(* IEC 61131-3 sources: volt/packages/volt-lsp-iec/test-corpus/bakon-nano/Device/Plc Logic/Application/POUs/HMI Functions, 3 files *)

(* ---- RecipeChoiceSelector.pou ---- *)
PROGRAM RecipeChoiceSelector
VAR
	nOldClmn1Choice : INT;
	nOldClmn2Choice : INT;
	bChoiceSetToZero : BOOL;
END_VAR

%LANGUAGE ST
/////////// First Column ////////////////////////////////////////////////////////////////////////////////
(*
Choices:
SlabRound = 1
SlabRound with fingers = 2
Tray = 3
*)

IF g_HMI_MachCommand.CMD.bNewRecipe AND NOT bChoiceSetToZero THEN
	g_sHMI_Recipe_Clmn1_Choice := 0;
	g_sHMI_Recipe_Clmn2_Choice := 0;
	g_sHMI_Recipe_Clmn2_Choice := 0;
	bChoiceSetToZero := TRUE;
END_IF
IF NOT(g_HMI_MachCommand.CMD.bNewRecipe) THEN
	bChoiceSetToZero := FALSE;
END_IF
g_sHMI_RcpClmns.clmn1.SlabRound := gProductOption.Prod_RoundQuatro
								OR gProductOption.Prod_SlabDiagonal
								OR gProductOption.Prod_SlabSquare
								OR gProductOption.Prod_SlabDouble
								OR gProductOption.Prod_SlabTriangle;

g_sHMI_RcpClmns.clmn1.SlabRoundFngrs := gProductOption.Prod_Round
									OR gProductOption.Prod_SlabSquareClamp;

g_sHMI_RcpClmns.clmn1.Tray := gProductOption.Prod_TraySquareDouble
								OR gProductOption.Prod_TraySquareLarge
								OR gProductOption.Prod_TraySquareSmall
								OR gProductOption.Prod_TraySquareTriple;

(*Reset choice for clmn 2 and 3 when 1 is changed *)
IF nOldClmn1Choice <> g_sHMI_Recipe_Clmn1_Choice THEN
	g_sHMI_Recipe_Clmn2_Choice := 0;
	g_sHMI_Recipe_Clmn3_Choice := 0;
	nOldClmn1Choice := g_sHMI_Recipe_Clmn1_Choice;
END_IF

//////////////////////////////////////////////////////////////////////////////////////////////////////////

/////////// Second Column ////////////////////////////////////////////////////////////////////////////////
(*
Choises:
Slab= 1
Slab with Fingers = 2
Round = 3
Round with fingers = 4
Tray Small = 5
Tray Large = 6
Tray double = 7
Tray Quadruple = 8
*)
g_sHMI_RcpClmns.clmn2.Slab := (gProductOption.Prod_SlabDiagonal
								OR gProductOption.Prod_SlabSquare
								OR gProductOption.Prod_SlabDouble
								OR gProductOption.Prod_SlabTriangle)
								AND (g_sHMI_Recipe_Clmn1_Choice = 1);

g_sHMI_RcpClmns.clmn2.SlabFingers := gProductOption.Prod_SlabSquareClamp AND (g_sHMI_Recipe_Clmn1_Choice = 2);

g_sHMI_RcpClmns.clmn2.Round := gProductOption.Prod_RoundQuatro AND (g_sHMI_Recipe_Clmn1_Choice = 1);

g_sHMI_RcpClmns.clmn2.RoundFingers := gProductOption.Prod_Round AND (g_sHMI_Recipe_Clmn1_Choice = 2 );

g_sHMI_RcpClmns.clmn2.TraySmall := gProductOption.Prod_TraySquareSmall AND (g_sHMI_Recipe_Clmn1_Choice = 3 );

g_sHMI_RcpClmns.clmn2.TrayLarge := gProductOption.Prod_TraySquareLarge AND (g_sHMI_Recipe_Clmn1_Choice = 3 );

g_sHMI_RcpClmns.clmn2.TrayQuadruple := gProductOption.Prod_TraySquareTriple AND (g_sHMI_Recipe_Clmn1_Choice = 3 );

g_sHMI_RcpClmns.clmn2.TrayDouble := gProductOption.Prod_TraySquareDouble AND (g_sHMI_Recipe_Clmn1_Choice = 3 );;

(*Reset choice for clmn 3 when 2 is changed *)
IF nOldClmn2Choice <> g_sHMI_Recipe_Clmn2_Choice THEN
	g_sHMI_Recipe_Clmn3_Choice := 0;
	nOldClmn2Choice := g_sHMI_Recipe_Clmn2_Choice;
END_IF
//////////////////////////////////////////////////////////////////////////////////////////////////////////

/////////// Third Column ////////////////////////////////////////////////////////////////////////////////
(*
Choices:
Square = 1
Round = 2
Diagonal = 3
*)
g_sHMI_RcpClmns.clmn3.Square := (gProductOption.Prod_SlabSquare
								OR gProductOption.Prod_TraySquareDouble
								OR gProductOption.Prod_TraySquareLarge
								OR gProductOption.Prod_TraySquareSmall
								OR gProductOption.Prod_TraySquareTriple
								OR gProductOption.Prod_SlabSquareClamp)
								AND (g_sHMI_Recipe_Clmn2_Choice <> 3)
								AND (g_sHMI_Recipe_Clmn2_Choice <> 4)
								AND (g_sHMI_Recipe_Clmn2_Choice <> 0);

g_sHMI_RcpClmns.clmn3.Triangle := (gProductOption.Prod_SlabSquare
								OR gProductOption.Prod_TraySquareLarge
								OR gProductOption.Prod_SlabSquareClamp)
								AND (g_sHMI_Recipe_Clmn2_Choice <> 2)
								AND (g_sHMI_Recipe_Clmn2_Choice <> 3)
								AND (g_sHMI_Recipe_Clmn2_Choice <> 4)
								AND (g_sHMI_Recipe_Clmn2_Choice <> 0);

g_sHMI_RcpClmns.clmn3.Diagonal := (gProductOption.Prod_SlabSquare
								OR gProductOption.Prod_SlabSquareClamp)
								AND (g_sHMI_Recipe_Clmn2_Choice <> 2)
								AND (g_sHMI_Recipe_Clmn2_Choice <> 3)
								AND (g_sHMI_Recipe_Clmn2_Choice <> 4)
								AND (g_sHMI_Recipe_Clmn2_Choice <> 0);

//////////////////////////////////////////////////////////////////////////////////////////////////////////

//////////select correct product in recipe////////////////////////////////////////////////////////////////
IF (g_sHMI_Recipe_Clmn1_Choice = 1) AND (g_sHMI_Recipe_Clmn2_Choice = 1) AND (g_sHMI_Recipe_Clmn3_Choice = 1) THEN
	g_HMI_RCP_Parameters_Visu.nProductType := Prod_Slab_Rectangle_1x1;
ELSIF (g_sHMI_Recipe_Clmn1_Choice = 1) AND (g_sHMI_Recipe_Clmn2_Choice = 1) AND (g_sHMI_Recipe_Clmn3_Choice = 2) THEN
	g_HMI_RCP_Parameters_Visu.nProductType := Prod_Slab_Triangle_1x1;
ELSIF (g_sHMI_Recipe_Clmn1_Choice = 1) AND (g_sHMI_Recipe_Clmn2_Choice = 1) AND (g_sHMI_Recipe_Clmn3_Choice = 3) THEN
	g_HMI_RCP_Parameters_Visu.nProductType := Prod_Slab_Diagonal_1x1;
ELSIF (g_sHMI_Recipe_Clmn1_Choice = 2) AND (g_sHMI_Recipe_Clmn2_Choice = 2) AND (g_sHMI_Recipe_Clmn3_Choice = 1) THEN
	g_HMI_RCP_Parameters_Visu.nProductType := Prod_Slab_Rectangle_1x1_Clamp;
ELSIF (g_sHMI_Recipe_Clmn1_Choice = 2) AND (g_sHMI_Recipe_Clmn2_Choice = 3) THEN
	g_HMI_RCP_Parameters_Visu.nProductType := Prod_Round_POC_2x1;
ELSIF (g_sHMI_Recipe_Clmn1_Choice = 2) AND (g_sHMI_Recipe_Clmn2_Choice = 4) THEN
	g_HMI_RCP_Parameters_Visu.nProductType := Prod_Round_POC_2x1;
ELSIF (g_sHMI_Recipe_Clmn1_Choice = 3) AND (g_sHMI_Recipe_Clmn2_Choice = 5) AND (g_sHMI_Recipe_Clmn3_Choice = 1)THEN
	g_HMI_RCP_Parameters_Visu.nProductType := Prod_Tray_Rectangle_1x2;
ELSIF (g_sHMI_Recipe_Clmn1_Choice = 3) AND (g_sHMI_Recipe_Clmn2_Choice = 6) AND (g_sHMI_Recipe_Clmn3_Choice = 1)THEN
	g_HMI_RCP_Parameters_Visu.nProductType := Prod_Tray_Rectangle_1x1;
	g_HMI_RCP_Parameters_Visu.bTrianglesInTray := FALSE;
ELSIF (g_sHMI_Recipe_Clmn1_Choice = 3) AND (g_sHMI_Recipe_Clmn2_Choice = 6) AND (g_sHMI_Recipe_Clmn3_Choice = 2)THEN
	g_HMI_RCP_Parameters_Visu.nProductType := Prod_Tray_Rectangle_1x1;
	g_HMI_RCP_Parameters_Visu.bTrianglesInTray := TRUE;
ELSIF (g_sHMI_Recipe_Clmn1_Choice = 3) AND (g_sHMI_Recipe_Clmn2_Choice = 7) THEN
	g_HMI_RCP_Parameters_Visu.nProductType := Prod_Tray_Rectangle_2x1;
ELSIF (g_sHMI_Recipe_Clmn1_Choice = 3) AND (g_sHMI_Recipe_Clmn2_Choice = 7) THEN
	g_HMI_RCP_Parameters_Visu.nProductType := Prod_Tray_Rectangle_1x4;
END_IF
//////////////////////////////////////////////////////////////////////////////////////////////////////////

END_PROGRAM

(* ---- VisuCutsHandler.pou ---- *)
PROGRAM VisuCutsHandler
VAR
	hCutLineCounter : INT;
	nOfVerCuts		: INT;
	vCutLineCounter : INT;
	nOfHorCuts		: INT;
	nOfDiagCuts		: INT;
	rCutAngle		: REAL;
	rCutX			: REAL;
	rCutY			: REAL;
	rLenghtCut		: REAL;
	c_PI			: REAL;
	nDeleteDiagFrom		: INT;
	nPiecesHor			: INT;
	nPiecesVer 			: INT;
	bTriangles			: BOOL;
	rProdSizeX			: REAL;
	rProdSizeY			: REAL;
	nActPartXsize		: INT;
	nActPartYsize		: INT;

	sLocalRecipeVar		: sMACH_RCP_Parameters;
END_VAR

%LANGUAGE ST
c_PI := 3.14159265359;
sLocalRecipeVar := g_HMI_RCP_Parameters_Visu;

nPiecesHor := sLocalRecipeVar.nPartsX;
nPiecesVer := sLocalRecipeVar.nPartsy;
bTriangles := (sLocalRecipeVar.nProductType = Prod_Slab_Triangle_1x1)
			OR ((sLocalRecipeVar.nProductType = Prod_Tray_Rectangle_1x1) AND sLocalRecipeVar.bTrianglesInTray);

(* ProductType = 0 = Slab Square *)
(* ProductType = 1 = Slab triangle *)
(* ProductType = 2 = Slab diagonal *)
(* ProductType = 3 = Round Cake *)
(* ProductType = 4 = Tray Square Small *)
(* ProductType = 5 = Tray Square Large *)

CASE sLocalRecipeVar.nProductType OF
	0,1,2:	rProdSizeX := sLocalRecipeVar.rProdLength_InX;
			rProdSizeY := sLocalRecipeVar.rProdLength_InY;

	3:	rProdSizeX := sLocalRecipeVar.rDiameterRound;
		rProdSizeY := sLocalRecipeVar.rDiameterRound;

	4:	rProdSizeX := g_HMI_MCH_Parameters.rProdLengthTraySmall_InX;
		rProdSizeY := g_HMI_MCH_Parameters.rProdLengthTraySmall_InY;

	5:	rProdSizeX := g_HMI_MCH_Parameters.rProdLengthTrayLarge_InX;
		rProdSizeY := g_HMI_MCH_Parameters.rProdLengthTrayLarge_InY;
END_CASE

nActPartXsize			:= REAL_TO_INT(rProdSizeX / nPiecesHor);
nActPartYsize			:= REAL_TO_INT(rProdSizeY / nPiecesVer);
g_HMI_RCP_ActPartSize := CONCAT(TO_STRING(nActPartXsize), ' x ');
g_HMI_RCP_ActPartSize := CONCAT(g_HMI_RCP_ActPartSize , TO_STRING(nActPartYsize));
g_HMI_RCP_ActPartSize := CONCAT(g_HMI_RCP_ActPartSize, ' mm');

(* Make waste visible when waste size is > 0, global function *)
g_sHMI_VisuCutsArray[1].visible := g_HMI_RCP_UseWasteLeft;
g_sHMI_VisuCutsArray[2].visible := g_HMI_RCP_UseWasteRight;
g_sHMI_VisuCutsArray[3].visible := g_HMI_RCP_UseWasteRear;
g_sHMI_VisuCutsArray[4].visible := g_HMI_RCP_UseWasteFront;

//trims op 0 als ze uit staan
		IF NOT(g_HMI_RCP_UseWasteLeft) THEN
			g_HMI_RCP_Parameters_Visu.rSizeTrimLeft := 0;
		END_IF

		IF NOT(g_HMI_RCP_UseWasteRight) THEN
			g_HMI_RCP_Parameters_Visu.rSizeTrimRight := 0;
		END_IF

		IF NOT(g_HMI_RCP_UseWasteFront) THEN
			g_HMI_RCP_Parameters_Visu.rSizeTrimFront := 0;
		END_IF

		IF NOT(g_HMI_RCP_UseWasteRear) THEN
			g_HMI_RCP_Parameters_Visu.rSizeTrimRear:= 0;
		END_IF

g_HMI_RCP_ShowRCPwastesettings := g_HMI_RCP_UseWasteLeft OR g_HMI_RCP_UseWasteRight OR g_HMI_RCP_UseWasteRear OR g_HMI_RCP_UseWasteFront;

(* Display vertial lines, for the horizontal pieces *)
(* line 5 - 50 are the lines for horizontal pieces*)
IF nPiecesHor > 1 THEN
	rCutX:=(512.0 / INT_TO_REAL(nPiecesHor));
	//calculate x pos for the lines. width of box is 512, offset is 10 and make visible if used
	nOfVerCuts := nPiecesHor - 1;
	FOR hCutLineCounter := 5 TO (5+(nOfVerCuts-1)) DO
		g_sHMI_VisuCutsArray[hCutLineCounter].xPos := CONCAT(TO_STRING((rCutX * (hCutLineCounter-4))+10), 'px');
		g_sHMI_VisuCutsArray[hCutLineCounter].visible := TRUE;
	END_FOR
		//make unused lines invisible
	FOR hCutLineCounter := (5+(nOfVerCuts)) TO 50 DO
		g_sHMI_VisuCutsArray[hCutLineCounter].visible := FALSE;
		g_sHMI_VisuCutsArray[hCutLineCounter].xPos := '0px';
	END_FOR
ELSE
	rCutX:=512.0;
	FOR hCutLineCounter := 5 TO 50 DO //dont display lines when the no of pieces is 0
		g_sHMI_VisuCutsArray[hCutLineCounter].visible := FALSE;
		g_sHMI_VisuCutsArray[hCutLineCounter].xPos := '0px';
	END_FOR
END_IF

(* Display horizontal lines, for the vertical pieces *)
(* line 51 - 95 are the lines for horizontal pieces*)
IF (nPiecesVer > 1) AND NOT(sLocalRecipeVar.nProductType = Prod_Slab_Diagonal_1x1) THEN
	//calculate y pos for the lines. height of box is 300 and make visible if used
	nOfHorCuts := nPiecesVer - 1;
	rCutY:=(300.0 / INT_TO_REAL(nPiecesVer));
	FOR vCutLineCounter := 51 TO (51+(nOfHorCuts-1)) DO
		g_sHMI_VisuCutsArray[vCutLineCounter].yPos := CONCAT(TO_STRING((rCutY * (vCutLineCounter-50))+10),'px');
		g_sHMI_VisuCutsArray[vCutLineCounter].visible := TRUE;
	END_FOR
		//make unused lines invisible
	FOR vCutLineCounter := (51+nOfHorCuts) TO 95 DO
		g_sHMI_VisuCutsArray[vCutLineCounter].visible := FALSE;
		g_sHMI_VisuCutsArray[vCutLineCounter].yPos := '0px';
	END_FOR
ELSE
	rCutY:= 300.0;
	FOR vCutLineCounter := 51 TO 95 DO //dont display lines when the no of pieces is 0 or diagonals are cut
		g_sHMI_VisuCutsArray[vCutLineCounter].visible := FALSE;
		g_sHMI_VisuCutsArray[vCutLineCounter].yPos := '0px';
	END_FOR
END_IF

(* Display diagonal lines, for triangles *)
(* line 100 - 150 are the lines for diagonal lines*)
IF bTriangles THEN
	rCutAngle := -((ATAN(rCuty/rCutX)) * (180/c_PI));
	nOfDiagCuts := nPiecesVer + (nPiecesHor-1);
	rLenghtCut := SQRT((rCutX * rCutX) + (rCuty * rCuty));
	FOR vCutLineCounter := 1 TO nOfDiagCuts DO
		g_sHMI_VisuCutsArray[vCutLineCounter+99].visible := TRUE;
		g_sHMI_VisuCutsArray[vCutLineCounter+99].rotation := rCutAngle;
		IF (nPiecesHor >= nPiecesVer) THEN
			IF vCutLineCounter <= (nPiecesVer) THEN
				g_sHMI_VisuCutsArray[vCutLineCounter+99].yPos := CONCAT(TO_STRING((rCutY * (vCutLineCounter))+10),'px');
				g_sHMI_VisuCutsArray[vCutLineCounter+99].xPos := CONCAT(TO_STRING(10), 'px');
				g_sHMI_VisuCutsArray[vCutLineCounter+99].length := CONCAT(TO_STRING(rLenghtCut * vCutLineCounter),'px');
			ELSIF (vCutLineCounter > (nPiecesVer)) AND (vCutLineCounter <= (nPiecesHor)) THEN
				g_sHMI_VisuCutsArray[vCutLineCounter+99].yPos := CONCAT(TO_STRING((300)+10),'px');
				g_sHMI_VisuCutsArray[vCutLineCounter+99].xPos := CONCAT(TO_STRING((rCutX * ((vCutLineCounter - (nPiecesVer)))+10)), 'px');
				g_sHMI_VisuCutsArray[vCutLineCounter+99].length := CONCAT(TO_STRING(rLenghtCut *nPiecesVer),'px');
			ELSE
				g_sHMI_VisuCutsArray[vCutLineCounter+99].visible := TRUE;
				g_sHMI_VisuCutsArray[vCutLineCounter+99].yPos := CONCAT(TO_STRING((300)+10),'px');
				g_sHMI_VisuCutsArray[vCutLineCounter+99].xPos := CONCAT(TO_STRING((rCutX * ((vCutLineCounter - (nPiecesVer)))+10)), 'px');
				g_sHMI_VisuCutsArray[vCutLineCounter+99].length :=  CONCAT(TO_STRING(rLenghtCut * (nPiecesHor-(vCutLineCounter - nPiecesVer))),'px');
			END_IF
		ELSE
			IF vCutLineCounter <= (nPiecesHor) THEN
				g_sHMI_VisuCutsArray[vCutLineCounter+99].yPos := CONCAT(TO_STRING((rCutY * (vCutLineCounter))+10),'px');
				g_sHMI_VisuCutsArray[vCutLineCounter+99].xPos := CONCAT(TO_STRING(10), 'px');
				g_sHMI_VisuCutsArray[vCutLineCounter+99].length := CONCAT(TO_STRING(rLenghtCut * vCutLineCounter),'px');
			ELSIF (vCutLineCounter > (nPiecesHor)) AND (vCutLineCounter <= (nPiecesVer)) THEN
				g_sHMI_VisuCutsArray[vCutLineCounter+99].yPos := CONCAT(TO_STRING((rCutY * (vCutLineCounter))+10),'px');
				g_sHMI_VisuCutsArray[vCutLineCounter+99].xPos := CONCAT(TO_STRING(10), 'px');
				g_sHMI_VisuCutsArray[vCutLineCounter+99].length := CONCAT(TO_STRING(rLenghtCut *nPiecesHor),'px');
			ELSE
				g_sHMI_VisuCutsArray[vCutLineCounter+99].yPos := CONCAT(TO_STRING((300)+10),'px');
				g_sHMI_VisuCutsArray[vCutLineCounter+99].xPos := CONCAT(TO_STRING((rCutX * ((vCutLineCounter - (nPiecesVer)))+10)), 'px');
				g_sHMI_VisuCutsArray[vCutLineCounter+99].length :=  CONCAT(TO_STRING(rLenghtCut * (nPiecesHor-(vCutLineCounter - nPiecesVer))),'px');
			END_IF
		END_IF
	END_FOR
	nDeleteDiagFrom := (100+nOfDiagCuts);
ELSE
	nDeleteDiagFrom := 100;
END_IF

//make all diagonal lines we don't need, invisible.
FOR vCutLineCounter := nDeleteDiagFrom TO 150 DO //dont display lines when the no of pieces is 0
	g_sHMI_VisuCutsArray[vCutLineCounter].visible := FALSE;
	g_sHMI_VisuCutsArray[vCutLineCounter].yPos := '0px';
	g_sHMI_VisuCutsArray[vCutLineCounter].xPos := '0px';
	g_sHMI_VisuCutsArray[vCutLineCounter].length := '0px';
	g_sHMI_VisuCutsArray[vCutLineCounter].rotation := 0.0;
END_FOR

END_PROGRAM

(* ---- VisuDashboardNotifications.pou ---- *)
PROGRAM VisuDashboardNotifications
VAR

END_VAR

%LANGUAGE ST
g_sHMI_DashboardNotifications.bCabinetError := g_sMACH.ERR.dwCat4_Error_a.6
											OR g_sMACH.ERR.dwCat4_Error_a.7
											OR g_sMACH.ERR.dwCat4_Error_a.8
											OR g_sMACH.ERR.dwCat4_Error_a.22;

g_sHMI_DashboardNotifications.bCleaningCilTimout := g_sMACH.ERR.dwCat4_Error_b.07
												OR g_sMACH.ERR.dwCat4_Error_b.08
												OR g_sMACH.ERR.dwCat4_Error_b.09;

g_sHMI_DashboardNotifications.bFrontRearmotorError := g_sMACH.ERR.dwCat4_Error_a.29
													OR g_sMACH.ERR.dwCat4_Error_a.30
													OR g_sMACH.ERR.dwCat4_Error_a.31
													OR g_sMACH.ERR.dwCat4_Error_a.9
													OR g_sMACH.ERR.dwCat4_Error_a.10
													OR g_sMACH.ERR.dwCat4_Error_a.13
													OR g_sMACH.ERR.dwCat4_Error_a.14
													OR g_sMACH.ERR.dwCat1_Error.6
													OR g_sMACH.ERR.dwCat1_Error.7;

g_sHMI_DashboardNotifications.bHeightCilTimout := g_sMACH.ERR.dwCat4_Error_b.14;

g_sHMI_DashboardNotifications.bHeightMotorError := g_sMACH.ERR.dwCat4_Error_a.11
												OR g_sMACH.ERR.dwCat4_Error_b.14;

g_sHMI_DashboardNotifications.bMainAirError := g_sMACH.ERR.dwCat4_Error_a.1;

g_sHMI_DashboardNotifications.bNSpanel := g_sMACH.ERR.dwCat4_Error_a.0;

g_sHMI_DashboardNotifications.bRmotorError := g_sMACH.ERR.dwCat4_Error_a.31
											OR g_sMACH.ERR.dwCat4_Error_a.12
											OR g_sMACH.ERR.dwCat1_Error.8;

g_sHMI_DashboardNotifications.bSafetyScreen := FALSE;

g_sHMI_DashboardNotifications.bUltrasonicError := g_sMACH.ERR.dwCat4_Error_a.5;

g_sHMI_DashboardNotifications.bUltrasonicWarning := g_sMACH.ERR.dwCat1_Error.10;

END_PROGRAM
